Staubli VAL3: OnF2.pgx

program OnF2()
  local num l_ni
  local bool l_bRes
begin
  //全部转换
  for l_ni=0 to size(sFileList)-1
    call OnePathConvert(sFolder,sFileList[l_ni],sOutputFolder,l_bRes)
    if !l_bRes
      popUpMsg(sFileList[l_ni]+"文件转换失败!")
      logMsg(sFileList[l_ni]+"文件转换失败!")
      wait(getKey()==278)
    endIf
  endFor
  popUpMsg("转换完成")
end
